FUNCTION TryConvert_DT_TO_DINT : BOOL
VAR_INPUT
	in : DT;
	out : REFERENCE TO DINT;
END_VAR

IF in > DatatypeLimits.MAX_VALUE_OF_DT_WHICH_CAN_BE_HELD_IN_A_DINT THEN
	RETURN;
END_IF

out := DT_TO_DINT(in);
TryConvert_DT_TO_DINT := TRUE;

END_FUNCTION

(* stored: Version 1.1.0.1, ProductVersion 3.1.4024.12
   POU TryConvert_DT_TO_DINT: Id {0eeb61a5-3ac7-4ddd-a033-4a2cf302a6bb}, SpecialFunc None *)
